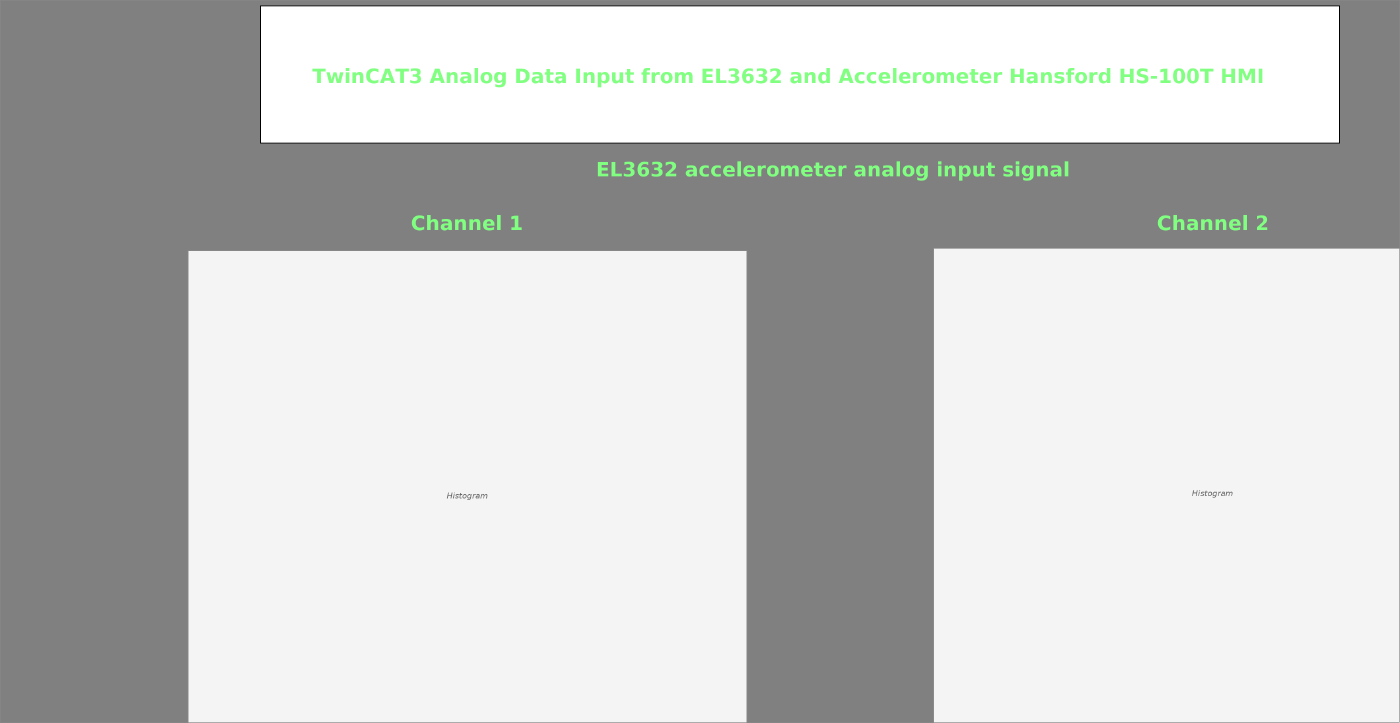
VISUALIZATION Visualization  // 1760x910, background image 
    Rectangle (327,7 1357x173)
    Label (764,153 575x120), "EL3632 accelerometer analog input signal"
    Textfield (459,1012 389x112), "Voltage: %.1f V", text variable: MAIN.EL3064.Voltage_1
    Meter360 (254,987 187x163), value: MAIN.EL3064.Voltage_1, style: Meter-Meter360-Gray, scale format: %.1f, scale 0..10
    Histogram (236,315 703x618), scale format: %.1f, scale -100..100
        p1518820177: MAIN.EL3632.Scaled_Ch1
        p102497268: MAIN.EL3632.Scaled_Ch1
        p788070771: ARRAY [1..10] OF REAL
    Label (358,20 1266x151), "TwinCAT3 Analog Data Input from EL3632 and Accelerometer Hansford HS-100T HMI"
    Histogram (1173,312 703x618), scale format: %.1f, scale -100..100
        p1518820177: MAIN.EL3632.Scaled_Ch2
        p102497268: MAIN.EL3632.Scaled_Ch2
        p788070771: ARRAY [1..10] OF REAL
    Label (468,235 238x91), "Channel 1"
    Label (1406,235 238x91), "Channel 2"
    Textfield (459,1208 389x112), "Voltage: %.1f V", text variable: MAIN.EL3064.Voltage_3
    Meter360 (257,1183 187x163), value: MAIN.EL3064.Voltage_3, style: Meter-Meter360-Gray, scale format: %.1f, scale 0..10
    Textfield (1268,1012 389x112), "Voltage: %.1f V", text variable: MAIN.EL3064.Voltage_2
    Meter360 (1063,987 187x163), value: MAIN.EL3064.Voltage_2, style: Meter-Meter360-Gray, scale format: %.1f, scale 0..10
    Textfield (1268,1208 389x112), "Voltage: %.1f V", text variable: MAIN.EL3064.Voltage_4
    Meter360 (1063,1183 187x163), value: MAIN.EL3064.Voltage_4, style: Meter-Meter360-Gray, scale format: %.1f, scale 0..10
    Label (25,897 575x120), "EL3064 Input Signal Voltage"
END_VISUALIZATION

(* stored: Version 1.1.0.1, ProductVersion 3.1.4024.16
   Visu Visualization: Id {5209e7c0-d504-401b-a552-d278f1762b3e} *)
